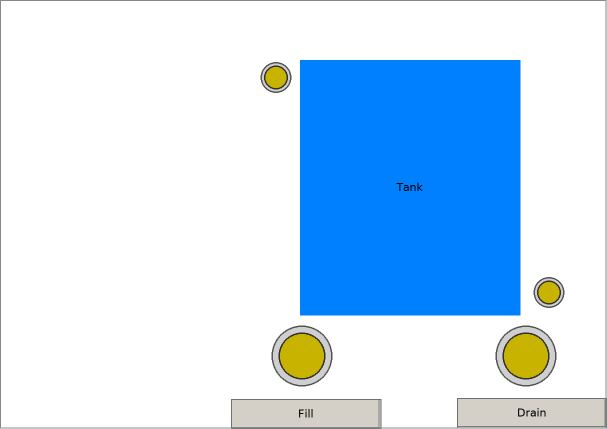
VISUALIZATION Visualization  // 607x429
    Lamp1 (267,321 70x70), variable: MAIN.fbLiquidTank.bFillLight, style: Lamp-Lamp1-Yellow
    Lamp1 (491,321 70x70), variable: MAIN.fbLiquidTank.bDrainLight, style: Lamp-Lamp1-Yellow
    Button (231,399 150x30), "Fill"
        tap MAIN.bFillButton
    Button (457,398 150x30), "Drain"
        tap MAIN.bDrainButton
    Rectangle (300,60 220x255), "Tank"
    Rectangle (300,145 220x85), "Tank", invisible if: NOT MAIN.fbLiquidTank.bVisMid
    Rectangle (300,60 220x85), invisible if: NOT MAIN.fbLiquidTank.bVisHigh
    Rectangle (300,230 220x85), invisible if: NOT MAIN.fbLiquidTank.bVisLow
    Lamp1 (258,58 36x39), variable: MAIN.fbLiquidTank.bHighSensor, style: Lamp-Lamp1-Yellow
    Lamp1 (531,273 36x39), variable: MAIN.fbLiquidTank.bLowSensor, style: Lamp-Lamp1-Yellow
END_VISUALIZATION

(* stored: Version 1.1.0.1, ProductVersion 3.1.4024.12
   Visu Visualization: Id {4bead43d-e8d8-4623-a897-cdf807b53a6c} *)
